// Mitsubishi GX Works2 project: 3u   PLC: FX3G

PROGRAM MAIN
VAR
  c_1 : c;
END_VAR
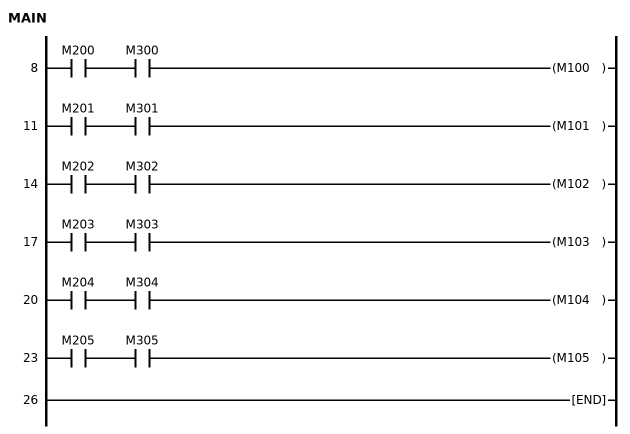
; FB BLK START c(c_1)
; FB START
; FB_NAME c
; INSTANCE_NAME c_1
; FB IN_B:ewq
; FB OUT_ewq:B
; FB END
; FB BLK END
8     LD      M200
      AND     M300
      OUT     M100
11    LD      M201
      AND     M301
      OUT     M101
14    LD      M202
      AND     M302
      OUT     M102
17    LD      M203
      AND     M303
      OUT     M103
20    LD      M204
      AND     M304
      OUT     M104
23    LD      M205
      AND     M305
      OUT     M105
26    END
END_PROGRAM

FUNCTION_BLOCK c
VAR_IN_OUT
  ewq : BOOL;
END_VAR
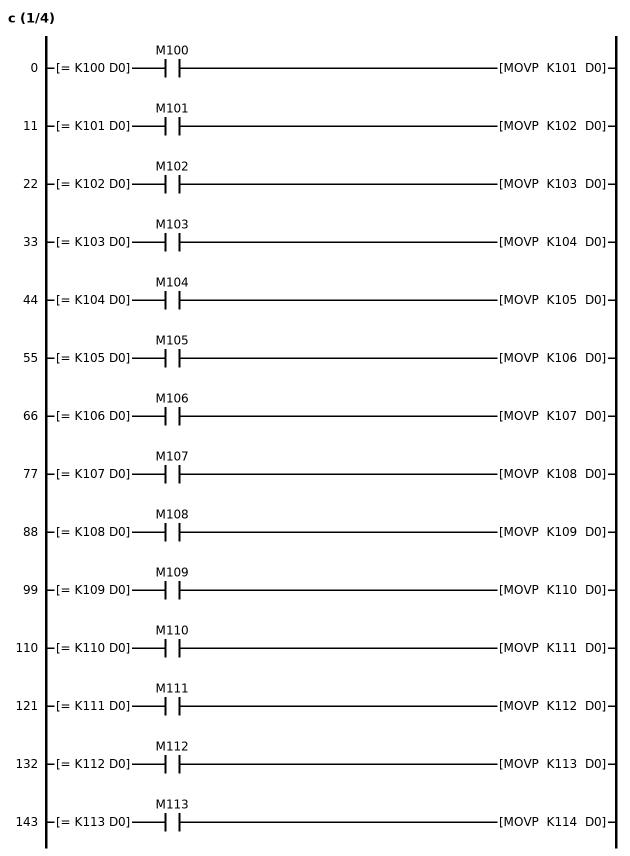
0     LD=     K100 D0
      AND     M100
      MOVP    K101 D0
11    LD=     K101 D0
      AND     M101
      MOVP    K102 D0
22    LD=     K102 D0
      AND     M102
      MOVP    K103 D0
33    LD=     K103 D0
      AND     M103
      MOVP    K104 D0
44    LD=     K104 D0
      AND     M104
      MOVP    K105 D0
55    LD=     K105 D0
      AND     M105
      MOVP    K106 D0
66    LD=     K106 D0
      AND     M106
      MOVP    K107 D0
77    LD=     K107 D0
      AND     M107
      MOVP    K108 D0
88    LD=     K108 D0
      AND     M108
      MOVP    K109 D0
99    LD=     K109 D0
      AND     M109
      MOVP    K110 D0
110   LD=     K110 D0
      AND     M110
      MOVP    K111 D0
121   LD=     K111 D0
      AND     M111
      MOVP    K112 D0
132   LD=     K112 D0
      AND     M112
      MOVP    K113 D0
143   LD=     K113 D0
      AND     M113
      MOVP    K114 D0
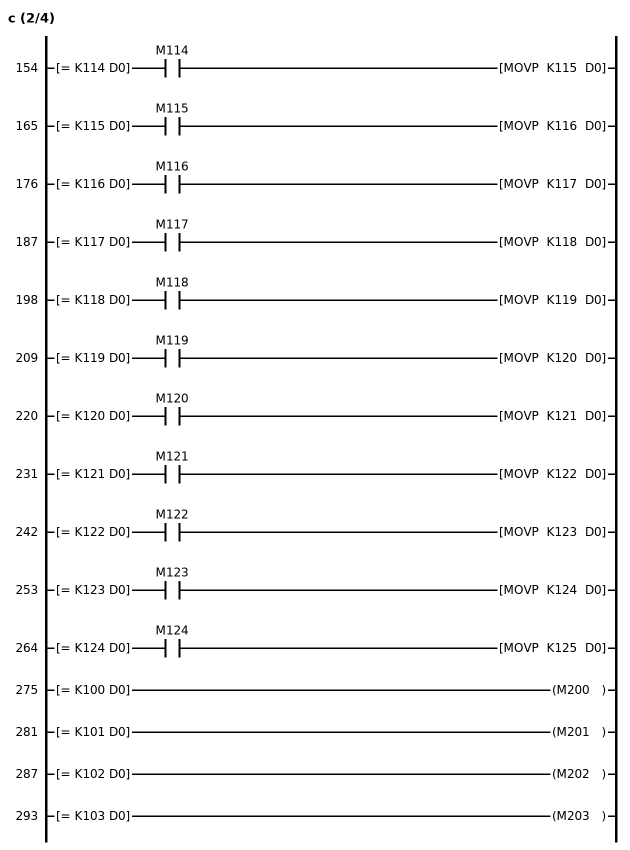
154   LD=     K114 D0
      AND     M114
      MOVP    K115 D0
165   LD=     K115 D0
      AND     M115
      MOVP    K116 D0
176   LD=     K116 D0
      AND     M116
      MOVP    K117 D0
187   LD=     K117 D0
      AND     M117
      MOVP    K118 D0
198   LD=     K118 D0
      AND     M118
      MOVP    K119 D0
209   LD=     K119 D0
      AND     M119
      MOVP    K120 D0
220   LD=     K120 D0
      AND     M120
      MOVP    K121 D0
231   LD=     K121 D0
      AND     M121
      MOVP    K122 D0
242   LD=     K122 D0
      AND     M122
      MOVP    K123 D0
253   LD=     K123 D0
      AND     M123
      MOVP    K124 D0
264   LD=     K124 D0
      AND     M124
      MOVP    K125 D0
275   LD=     K100 D0
      OUT     M200
281   LD=     K101 D0
      OUT     M201
287   LD=     K102 D0
      OUT     M202
293   LD=     K103 D0
      OUT     M203
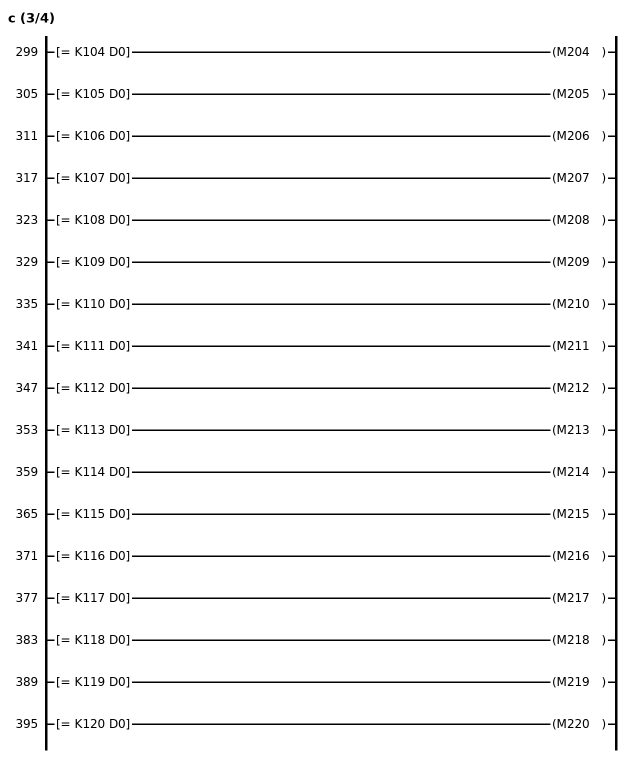
299   LD=     K104 D0
      OUT     M204
305   LD=     K105 D0
      OUT     M205
311   LD=     K106 D0
      OUT     M206
317   LD=     K107 D0
      OUT     M207
323   LD=     K108 D0
      OUT     M208
329   LD=     K109 D0
      OUT     M209
335   LD=     K110 D0
      OUT     M210
341   LD=     K111 D0
      OUT     M211
347   LD=     K112 D0
      OUT     M212
353   LD=     K113 D0
      OUT     M213
359   LD=     K114 D0
      OUT     M214
365   LD=     K115 D0
      OUT     M215
371   LD=     K116 D0
      OUT     M216
377   LD=     K117 D0
      OUT     M217
383   LD=     K118 D0
      OUT     M218
389   LD=     K119 D0
      OUT     M219
395   LD=     K120 D0
      OUT     M220
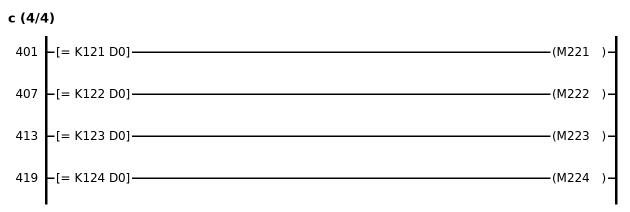
401   LD=     K121 D0
      OUT     M221
407   LD=     K122 D0
      OUT     M222
413   LD=     K123 D0
      OUT     M223
419   LD=     K124 D0
      OUT     M224
END_FUNCTION_BLOCK
